Staubli VAL3: initvis.pgx

program initvis(bool& x_bResult[])
  local bool l_bResult
begin
  // Initialize cognex communication library
  call cam:init()
  x_bResult=true
  clearBuffer(skVision)
  put("logging in to camera...")
  // log in to camera using socket cognex1 and return a handle in hCamTable
  //
  call cam:login(skVision,"admin","",hCamTable,l_bResult)
  if l_bResult
    putln("ok")
  else
    call cam:getErrorMessage(hCamTable,strError)
    putln("failed: "+strError)
    x_bResult=false
  endIf
  call cam:getOnline(hCamTable,l_bResult)
  if !l_bResult
    putln("Camera is not online")
    x_bResult=false
  endIf
end
